INTERFACE I_DeserializerGarbageCollector EXTENDS __SYSTEM.IQueryInterface

METHOD PUBLIC Deregister
VAR_INPUT
	Deserializer : I_Deserializer;
END_VAR
END_METHOD

METHOD PUBLIC Register
VAR_INPUT
	Deserializer : I_Deserializer;
END_VAR
END_METHOD

END_INTERFACE

(* stored: Version 1.1.0.1, ProductVersion 3.1.4024.12
   Itf I_DeserializerGarbageCollector: Id {3ba5eb31-a337-00b9-3e08-84cebca0c801}
   Method Deregister: Id {bff3cb11-fe5c-0289-0fe2-5f6c012703e4}
   Method Register: Id {0a568702-a564-035e-11c9-2fb5256ab6c9} *)
